{attribute 'qualified_only'}
{attribute 'strict'}
{attribute 'to_string'}
TYPE E_FsmState :
(
	ERR       := 0,
	INIT      := 1,
	STAT      := 2, 
	STAT_TR   := 3,
	NOM_LEV   := 4,
	INTER_TR  := 5,
	END_TR 	  := 6
);
END_TYPE

(* stored: Version 1.1.0.1, ProductVersion 3.1.4024.10
   DUT E_FsmState: Id {58d95daf-7d74-49ae-8fa0-ac8cbb3f5a9c} *)
